(* LS Electric XG5000 project: GS20_Mbtcp *)
(* GS20 modbus tcp setup *)
(* PLC LSPLC *)
(* module base 0 slot 0: Input/Output Module:XEM-DN/DP32HP (DC 24V Input, Transistor Output, 32 Contacts) *)
(* module base 0 slot 1: Internal Positioning:XBF-PO06E (Open Collector Type, 6 Axis) *)

(* Comments on direct variables
%MW0	2100_StatusMon1
%MW1	2101_StatusMon2
%MW2	2102_FreqCommand
%MW3	2103_OutputFreq
%MW4	2104_OutputCurr
%MW5	2105_DCBusVolt
%MW6	2106_OutputVolt
%MW7	2107_MultiSpeed
%MW8	2108_Reserved
%MW9	2109_DigitalInputCounter
%MW20	2000_ControlWord
%MW21	2001_ControlFreq
%MW22	2002_ControlReset
*)

PROGRAM NewProgram (* task: Scan Program *)

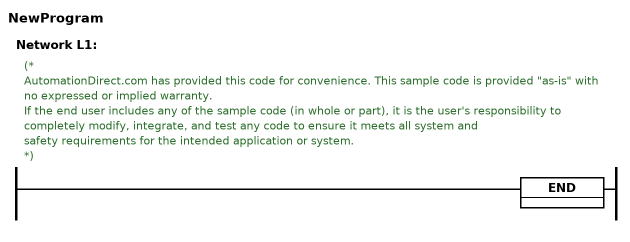
(* ( * / AutomationDirect.com has provided this code for convenience. This sample code is provided "as-is" with no expressed or implied warranty. / If the end user includes any of the sample code (in whole or part), it is the user's responsibility to completely modify, integrate, and test any code to ensure it meets all system and / safety requirements for the intended application or system. / * ) *)
(* Rung L1 *)
END();
END_PROGRAM